FUNCTION_BLOCK comandoAutomatico (* Basic Function Block Type *)
  (* Standard: 61499-2 *)
  (* Version 0.0, 01/03/2026, Template *)
  PACKAGE Hidryco.HidrycoLib;
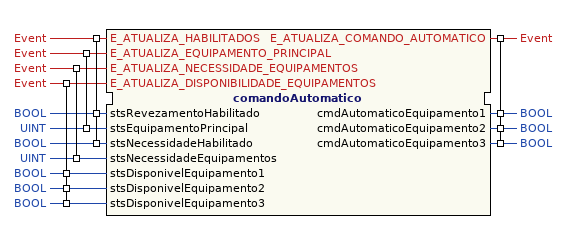
  EVENT_INPUT
    E_ATUALIZA_HABILITADOS WITH stsRevezamentoHabilitado, stsNecessidadeHabilitado;
    E_ATUALIZA_EQUIPAMENTO_PRINCIPAL WITH stsEquipamentoPrincipal;
    E_ATUALIZA_NECESSIDADE_EQUIPAMENTOS WITH stsNecessidadeEquipamentos;
    E_ATUALIZA_DISPONIBILIDADE_EQUIPAMENTOS WITH stsDisponivelEquipamento1, stsDisponivelEquipamento2, stsDisponivelEquipamento3;
  END_EVENT
  EVENT_OUTPUT
    E_ATUALIZA_COMANDO_AUTOMATICO WITH cmdAutomaticoEquipamento1, cmdAutomaticoEquipamento2, cmdAutomaticoEquipamento3;
  END_EVENT
  VAR_INPUT
    stsRevezamentoHabilitado : BOOL;
    stsEquipamentoPrincipal : UINT;
    stsNecessidadeHabilitado : BOOL;
    stsNecessidadeEquipamentos : UINT;
    stsDisponivelEquipamento1 : BOOL;
    stsDisponivelEquipamento2 : BOOL;
    stsDisponivelEquipamento3 : BOOL;
  END_VAR
  VAR_OUTPUT
    cmdAutomaticoEquipamento1 : BOOL;
    cmdAutomaticoEquipamento2 : BOOL;
    cmdAutomaticoEquipamento3 : BOOL;
  END_VAR
  VAR
    equipamentosDisponiveis : INT;
  END_VAR
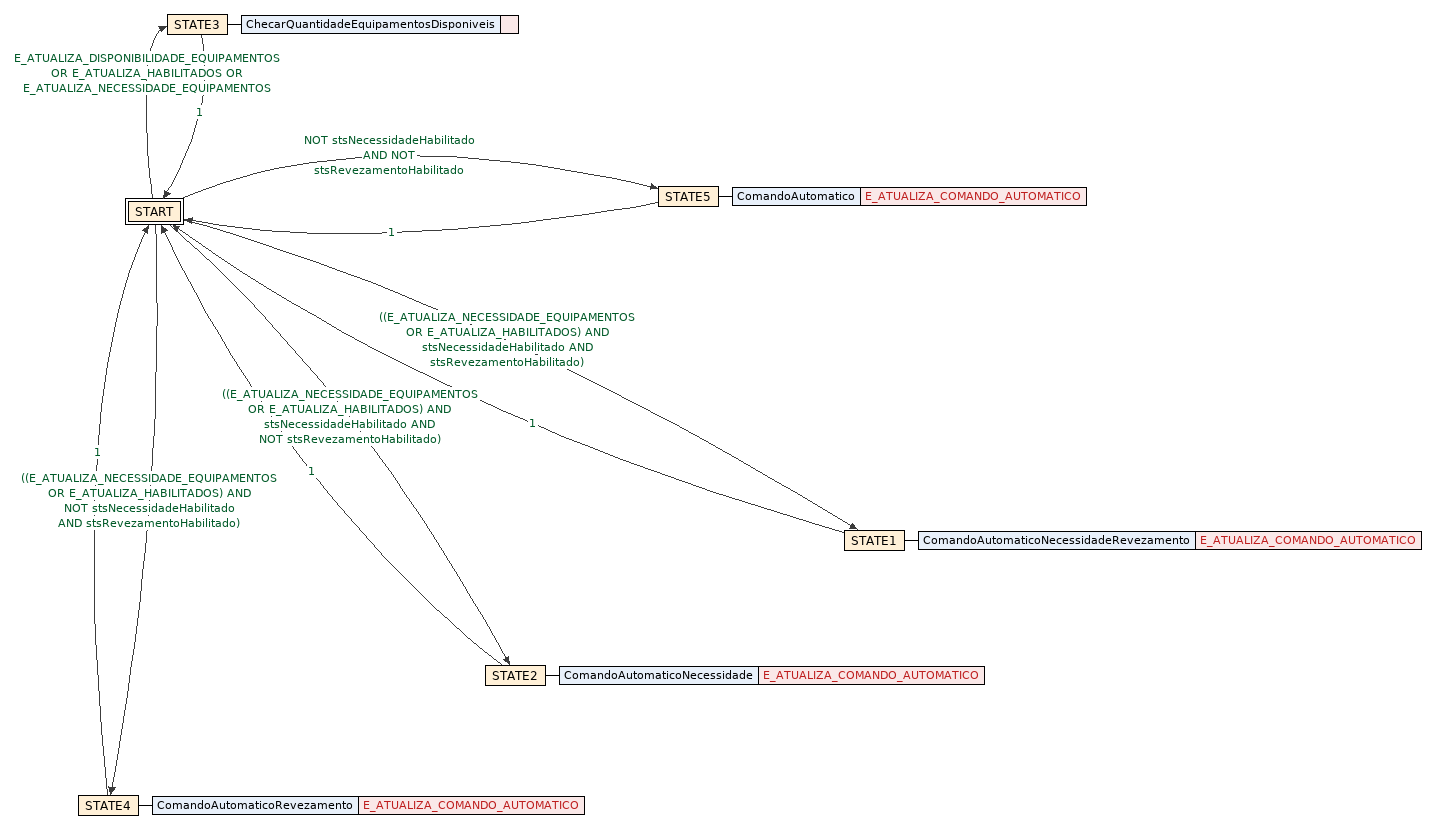
  EC_STATES
    START; (* Initial State *)
    STATE1 : ComandoAutomaticoNecessidadeRevezamento -> E_ATUALIZA_COMANDO_AUTOMATICO;
    STATE2 : ComandoAutomaticoNecessidade -> E_ATUALIZA_COMANDO_AUTOMATICO;
    STATE3 : ChecarQuantidadeEquipamentosDisponiveis;
    STATE4 : ComandoAutomaticoRevezamento -> E_ATUALIZA_COMANDO_AUTOMATICO;
    STATE5 : ComandoAutomatico -> E_ATUALIZA_COMANDO_AUTOMATICO;
  END_STATES
  EC_TRANSITIONS
    START TO STATE3 := E_ATUALIZA_DISPONIBILIDADE_EQUIPAMENTOS OR E_ATUALIZA_HABILITADOS OR E_ATUALIZA_NECESSIDADE_EQUIPAMENTOS;
    STATE3 TO START := 1;
    START TO STATE1 := ((E_ATUALIZA_NECESSIDADE_EQUIPAMENTOS OR E_ATUALIZA_HABILITADOS) AND stsNecessidadeHabilitado AND stsRevezamentoHabilitado);
    STATE1 TO START := 1;
    START TO STATE2 := ((E_ATUALIZA_NECESSIDADE_EQUIPAMENTOS OR E_ATUALIZA_HABILITADOS) AND stsNecessidadeHabilitado AND NOT stsRevezamentoHabilitado);
    STATE2 TO START := 1;
    START TO STATE4 := ((E_ATUALIZA_NECESSIDADE_EQUIPAMENTOS OR E_ATUALIZA_HABILITADOS) AND NOT stsNecessidadeHabilitado AND stsRevezamentoHabilitado);
    STATE4 TO START := 1;
    START TO STATE5 := NOT stsNecessidadeHabilitado AND NOT stsRevezamentoHabilitado;
    STATE5 TO START := 1;
  END_TRANSITIONS
  ALGORITHM ComandoAutomaticoNecessidadeRevezamento IN ST:
IF (stsNecessidadeEquipamentos = 1 OR (equipamentosDisponiveis = 1 AND stsNecessidadeEquipamentos > 0)) THEN
	cmdAutomaticoEquipamento1 := (stsEquipamentoPrincipal = 1);
	cmdAutomaticoEquipamento2 := (stsEquipamentoPrincipal = 2);
	cmdAutomaticoEquipamento3 := (stsEquipamentoPrincipal = 3);

ELSIF (stsNecessidadeEquipamentos = 2 AND equipamentosDisponiveis > 1) THEN
	cmdAutomaticoEquipamento1 := (stsDisponivelEquipamento1 AND ((stsEquipamentoPrincipal = 1) OR (stsEquipamentoPrincipal = 2 AND (NOT stsDisponivelEquipamento3)) OR (stsEquipamentoPrincipal = 3)));
	cmdAutomaticoEquipamento2 := (stsDisponivelEquipamento2 AND ((stsEquipamentoPrincipal = 2) OR (stsEquipamentoPrincipal = 3 AND (NOT stsDisponivelEquipamento1)) OR (stsEquipamentoPrincipal = 1)));
	cmdAutomaticoEquipamento3 := (stsDisponivelEquipamento3 AND ((stsEquipamentoPrincipal = 3) OR (stsEquipamentoPrincipal = 1 AND (NOT stsDisponivelEquipamento2)) OR (stsEquipamentoPrincipal = 2)));

ELSE
	cmdAutomaticoEquipamento1 := FALSE;
	cmdAutomaticoEquipamento2 := FALSE;
	cmdAutomaticoEquipamento3 := FALSE;
END_IF;
;
  END_ALGORITHM
  ALGORITHM ComandoAutomaticoNecessidade IN ST:
IF stsNecessidadeEquipamentos = 1 OR (equipamentosDisponiveis = 1 AND stsNecessidadeEquipamentos > 0) THEN
	cmdAutomaticoEquipamento1 := (stsDisponivelEquipamento1);
	cmdAutomaticoEquipamento2 := (stsDisponivelEquipamento2 AND NOT stsDisponivelEquipamento1);
	cmdAutomaticoEquipamento3 := (stsDisponivelEquipamento3 AND (NOT stsDisponivelEquipamento1) AND (NOT stsDisponivelEquipamento2));

ELSIF (stsNecessidadeEquipamentos = 2 AND equipamentosDisponiveis > 1) THEN
	cmdAutomaticoEquipamento1 := (stsDisponivelEquipamento1);
	cmdAutomaticoEquipamento2 := (stsDisponivelEquipamento2);
	cmdAutomaticoEquipamento3 := (NOT stsDisponivelEquipamento1) OR (NOT stsDisponivelEquipamento2);

ELSE
	cmdAutomaticoEquipamento1 := FALSE;
	cmdAutomaticoEquipamento2 := FALSE;
	cmdAutomaticoEquipamento3 := FALSE;
END_IF;
;
  END_ALGORITHM
  ALGORITHM ChecarQuantidadeEquipamentosDisponiveis IN ST:
equipamentosDisponiveis := BOOL_TO_INT(stsDisponivelEquipamento1) + BOOL_TO_INT(stsDisponivelEquipamento2) +  BOOL_TO_INT(stsDisponivelEquipamento3);
;
  END_ALGORITHM
  ALGORITHM ComandoAutomaticoRevezamento IN ST:
IF stsEquipamentoPrincipal > 0 THEN
	cmdAutomaticoEquipamento1 := (stsEquipamentoPrincipal = 1);
	cmdAutomaticoEquipamento2 := (stsEquipamentoPrincipal = 2);
	cmdAutomaticoEquipamento3 := (stsEquipamentoPrincipal = 3);
ELSE
	cmdAutomaticoEquipamento1 := FALSE;
	cmdAutomaticoEquipamento2 := FALSE;
	cmdAutomaticoEquipamento3 := FALSE;
END_IF;
;
  END_ALGORITHM
  ALGORITHM ComandoAutomatico IN ST:
cmdAutomaticoEquipamento1 := (stsDisponivelEquipamento1);
cmdAutomaticoEquipamento2 := (stsDisponivelEquipamento2);
cmdAutomaticoEquipamento3 := (stsDisponivelEquipamento3);
;
  END_ALGORITHM
END_FUNCTION_BLOCK
